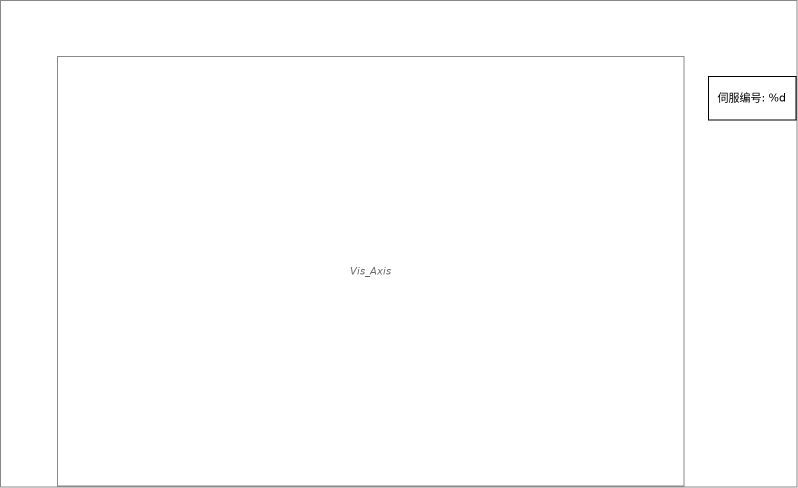
VISUALIZATION Vis_RealAxis  // 798x488
    Frame (57,56 627x430)
        shows Vis_Axis(Axis := MotionControl.Vis_RealAxisRef)
    Rectangle (708,76 88x44), "伺服编号: %d", text variable: MotionControl.Vis_RealAxisNoRef
        OnMouseClick: write the text variable via Default
END_VISUALIZATION

(* stored: Version 1.1.0.1, ProductVersion 3.1.4022.16
   Visu Vis_RealAxis: Id {8bfc6271-ad79-4c1f-8b6c-e6ac768ad0ef} *)
